// TIA Portal V19 export
DATA_BLOCK "DEBUG_MES_Send_Msg_1XX"   // DB15
// stored: MemoryReserve 100
   VAR
      MSG101 : Struct
         ABILITA_FC : Bool;
         EXE : Bool;
         RETVAL : DInt;
         Err { ExternalAccessible := 'False'; ExternalVisible := 'False'; ExternalWritable := 'False'} : "MES_Err_&_Msg";
      END_STRUCT;
      MSG102 : Struct
         ABILITA_FC : Bool;
         EXE : Bool;
         RETVAL : DInt;
         Err { ExternalAccessible := 'False'; ExternalVisible := 'False'; ExternalWritable := 'False'} : "MES_Err_&_Msg";
         MSG102 : Struct
            ABILITA_FC : Bool;
            EXE : Bool;
            RETVAL : DInt;
            Err { ExternalAccessible := 'False'; ExternalVisible := 'False'; ExternalWritable := 'False'} : "MES_Err_&_Msg";
         END_STRUCT;
      END_STRUCT;
      TEST_FUN_BUFFER : Struct
         ABILITA_FC : Bool;
         RETVAL : DInt;
         lastId : DInt;   // id ultimo messaggio inviato
         Index : Int;   // contatore messaggi da inviare
         Msg : "MES_Msg";
         Evaluate_FULL : Bool;
         ClearGap : Bool;
         Push : Bool;
         Pop : Bool;
      END_STRUCT;
   END_VAR
BEGIN
END_DATA_BLOCK
